{attribute 'qualified_only'}
{attribute 'strict'}
TYPE MC_COMBINE_MODE :
(
	enum_member := 0
);
END_TYPE

(* stored: Version 1.1.0.1, ProductVersion 3.1.4024.11
   DUT MC_COMBINE_MODE: Id {69ea87cd-8db4-4866-bafe-ed6e2613110d} *)
